TYPE ST_StatusBasic :
STRUCT
    Busy	:BOOL;	// TRUE : Process is running
    Done	:BOOL;	// TRUE : Process is done
    Error	:BOOL;	// TRUE : Process has error
	//ErrorID :UINT;
	Status : T_MaxString; // Show the error msg
END_STRUCT
END_TYPE

(* stored: Version 1.1.0.1, ProductVersion 3.1.4024.13
   DUT ST_StatusBasic: Id {fedf47fd-8b74-4b3e-bffa-b63532a03ef9} *)
